{attribute 'GeneratedUsingTerminal: EP7342-0002-0016'}
{attribute addProperty BoxType "EP7342-0002-0016"}
{attribute addProperty Id "ControlAT %Q*Control_F189B7373Set_counter_valueAT %Q*UINT2"}
{attribute addProperty CRC "780319811"}
{attribute addProperty Size "5"}
TYPE ENC_Control_compact_Channel_2E82BC43 EXTENDS OutputBase_10CEE7DE :
STRUCT
	{attribute addProperty Name "Control"}
	Control AT %Q* : Control_F189B737;
	{attribute addProperty Name "Set_counter_value"}
	Set_counter_value AT %Q* : UINT;
END_STRUCT
END_TYPE

(* stored: Version 1.2.0.0, ProductVersion 3.1.4024.9
   DUT ENC_Control_compact_Channel_2E82BC43: Id {3499fa5c-d140-4d0b-b2c9-30bc7645a55d} *)
